# B&R Automation Studio project Huitong_FrontEval
Automation Studio 6.5.0.306; technology packages: mappView 6.5.0, OpcUaCs 6.0.0

## Configuration Config1

CPU X20CP3687X, AutomationRuntime 6.5.1, Build 11.3.0, Vc 6.0.0

### Task classes (Cpu.sw)
```
Cyclic#2:
  MidTrans <- Middleware.MidTrans.prg
Cyclic#4:
  SVG <- SVG.prg
Binaries: FWRules, mvLoader, mvConfig, udbdef, TCData, iomap, UaCsConfig, BRRole, sysconf, asfw, User, arconfig, ashwd, Role, ashwac
Libraries: AsBrStr, ArSsl, FileIO, AsARCfg, runtime, standard
```

### Hardware
```
X20CP3687X : X20CP3687X v1.9.0.0
  Connector IF2:
    ActivateDevice = 1
    Mode = Manual
    InternetAddress = 192.168.50.233
    SubnetMask = 255.255.255.0
    ActivateSnmp = 2
  ConfigurationID = Huitong_FrontEval_Config1
  Simulation = 1
  FileDevice1
  FileDeviceName1 = USER
  FileDevicePath1 = USER_PATH
  ActivateFtpServer = 1
  FTPProtocol = 1
  FtpUser1
  FtpUsername1 = br
  FtpUserPassword1 = Vr55dmG4DfTukFxBuZ2vPJZUQAb9yWCctBfVGawW8Bk=  // 123456
  FtpUserSalt1 = kenBVaZZ
  FTPAccessRight1 = 0
  ActivateWebServer = 1
  WebServerProtocol = 1
  WebServerPort = 82
  WebServerWebDir = CFCARD\WEBROOT\
  WebServerStartPage = color01.html
  WebServerAspActivate = 1
  WebServerAspReadOnly = 0
  ActivateSdm = 1
```

## Configuration x1685

CPU X20CP1685, AutomationRuntime 6.5.1, Build 11.3.0, Vc 6.0.0

### Task classes (Cpu.sw)
```
Cyclic#2:
  MidTrans <- Middleware.MidTrans.prg
Cyclic#3:
  LQR <- LQR.prg
Cyclic#4:
  SVG <- SVG.prg
Cyclic#5:
  HmiBridge <- Middleware.HmiBridge.prg
Binaries: FWRules, mvLoader, mvConfig, udbdef, TCData, iomap, UaCsConfig, BRRole, sysconf, asfw, User, arconfig, ashwd, Role, ashwac
Libraries: AsBrStr, ArSsl, FileIO, AsARCfg, runtime, standard
```

### Hardware
```
X20CP1685 : X20CP1685 v1.9.0.0
  Connector IF2:
    ActivateDevice = 1
    Mode = Manual
    InternetAddress = 192.168.50.222
    SubnetMask = 255.255.255.0
    ActivateSnmp = 2
  Connector IF3:
    CycleTime = 400
  ConfigurationID = Huitong_FrontEval_Config1
  FileDevice1
  FileDeviceName1 = USER
  FileDevicePath1 = USER_PATH
  ActivateFtpServer = 1
  FTPProtocol = 1
  FtpUser1
  FtpUsername1 = br
  FtpUserPassword1 = Vr55dmG4DfTukFxBuZ2vPJZUQAb9yWCctBfVGawW8Bk=  // 123456
  FtpUserSalt1 = kenBVaZZ
  FTPAccessRight1 = 0
  ActivateWebServer = 1
  WebServerProtocol = 1
  WebServerPort = 82
  WebServerWebDir = CFCARD\WEBROOT\
  WebServerStartPage = color01.html
  WebServerAspActivate = 1
  WebServerAspReadOnly = 0
  ActivateSdm = 1
```

## Configuration x3687x

### Task classes (Cpu.sw)
```
Cyclic#2:
  MidTrans <- Middleware.MidTrans.prg
Cyclic#3:
  LQR <- LQR.prg
Cyclic#4:
  SVG <- SVG.prg
Binaries: FWRules, mvLoader, mvConfig, udbdef, TCData, iomap, UaCsConfig, BRRole, sysconf, asfw, User, arconfig, ashwd, Role, ashwac
Libraries: AsBrStr, ArSsl, FileIO, AsARCfg, runtime, standard
```

### Hardware
```
X20CP3687X : X20CP3687X v1.9.0.0
  Connector IF2:
    ActivateDevice = 1
    Mode = Manual
    InternetAddress = 192.168.50.233
    SubnetMask = 255.255.255.0
    ActivateSnmp = 2
  ConfigurationID = Huitong_FrontEval_Config1
  FileDevice1
  FileDeviceName1 = USER
  FileDevicePath1 = USER_PATH
  ActivateFtpServer = 1
  FTPProtocol = 1
  FtpUser1
  FtpUsername1 = br
  FtpUserPassword1 = Vr55dmG4DfTukFxBuZ2vPJZUQAb9yWCctBfVGawW8Bk=  // 123456
  FtpUserSalt1 = kenBVaZZ
  FTPAccessRight1 = 0
  ActivateWebServer = 1
  WebServerProtocol = 1
  WebServerPort = 82
  WebServerWebDir = CFCARD\WEBROOT\
  WebServerStartPage = color01.html
  WebServerAspActivate = 1
  WebServerAspReadOnly = 0
  ActivateSdm = 1
```

## Logical view

Binary libraries used (declarations not repeated): operator, runtime, AsIecCon, AsBrStr, AsARCfg, standard

### Package Logical/Libraries - Global libraries

- Visualisation Logical/mappView (not shown)

### Program Logical/Middleware/MidTrans (ANSIC)

#### Main.c - Init, cyclic, exit code
```c
#include <bur/plctypes.h>

#include <stdio.h>
#include <stdint.h>
#include <string.h>
#include <math.h>

#include "Function.h"

#define SIN_DATA_LENGTH 1000
#define SIN_AMPLITUDE 127.5
#define SIN_OFFSET 127.5
#define MAX_UDINT 4294967295U

#ifdef _DEFAULT_INCLUDES
	#include <AsDefault.h>
#endif

void _INIT ProgramInit(void)
{
	gstHmi.stInputs.diLockBoxWidth = 40;
	gstMainInface.stFromMain.diSImage = 600;
	gstMainInface.stToMain.usiActivePU = 0;
	brsstrcpy((UDINT)gstHmi.stConfig.strPuChartAdr, (UDINT)&"http://");

	/********************计算IP**************************/
	fbCfgGetIPAddr.enable = 1;
	fbCfgGetIPAddr.pDevice = (UDINT)&"IF2";
	fbCfgGetIPAddr.pIPAddr = (UDINT)strTemp;
	fbCfgGetIPAddr.Len = sizeof(strTemp);
	CfgGetIPAddr(&fbCfgGetIPAddr);

	brsstrcat((UDINT)gstHmi.stConfig.strPuChartAdr, (UDINT)strTemp);
	bSimTemp = 1;
}

void _CYCLIC ProgramCyclic(void)
{
	/**********************************以下为临时程序***************************************************/
	if(1 == bSimTemp) {
		/********************** 模拟仿真数据生成 ***************************/
		if(0 == stOldHmiInput.bRefreshSimData && 1 == gstHmi.stInputs.bRefreshSimData) {
			for(udiIdx = 0; udiIdx < ST_DATA_LEN; udiIdx++) {
				rSinValue = sin(2.0 * 3.14159265358979 * (REAL)(udiSinPhase + udiIdx) / 1000.0);
				gstMainInface.stFromMain.usiDataST1[udiIdx] = (USINT)(rSinValue * SIN_AMPLITUDE + SIN_OFFSET);

				rSinValue = sin(2.0 * 3.14159265358979 * (REAL)(udiSinPhase + udiIdx + 250) / 1000.0);
				gstMainInface.stFromMain.usiDataST2[udiIdx] = (USINT)(rSinValue * SIN_AMPLITUDE + SIN_OFFSET);

				rSinValue = sin(2.0 * 3.14159265358979 * (REAL)(udiSinPhase + udiIdx + 500) / 1000.0);
				gstMainInface.stFromMain.usiDataST3[udiIdx] = (USINT)(rSinValue * SIN_AMPLITUDE + SIN_OFFSET);

				rSinValue = sin(2.0 * 3.14159265358979 * (REAL)(udiSinPhase + udiIdx + 750) / 1000.0);
				gstMainInface.stFromMain.usiDataST4[udiIdx] = (USINT)(rSinValue * SIN_AMPLITUDE + SIN_OFFSET);

				rSinValue = sin(2.0 * 3.14159265358979 * (REAL)(udiSinPhase + udiIdx + 1000) / 1000.0);
				gstMainInface.stFromMain.usiDataST5[udiIdx] = (USINT)(rSinValue * SIN_AMPLITUDE + SIN_OFFSET);

				rSinValue = sin(2.0 * 3.14159265358979 * (REAL)(udiSinPhase + udiIdx + 1250) / 1000.0);
				gstMainInface.stFromMain.usiDataST6[udiIdx] = (USINT)(rSinValue * SIN_AMPLITUDE + SIN_OFFSET);
			}
		}

		if(0 == stOldHmiInput.bMoveCurveLeft && 1 == gstHmi.stInputs.bMoveCurveLeft) {
			for(udiIdx = 0; udiIdx < ST_DATA_LEN; udiIdx++) {
				rSinValue = sin(2.0 * 3.14159265358979 * (REAL)(udiSinPhase + udiIdx) / 1000.0);
				gstMainInface.stFromMain.usiDataST1[udiIdx] = (USINT)(rSinValue * SIN_AMPLITUDE + SIN_OFFSET);

				rSinValue = sin(2.0 * 3.14159265358979 * (REAL)(udiSinPhase + udiIdx + 250) / 1000.0);
				gstMainInface.stFromMain.usiDataST2[udiIdx] = (USINT)(rSinValue * SIN_AMPLITUDE + SIN_OFFSET);

				rSinValue = sin(2.0 * 3.14159265358979 * (REAL)(udiSinPhase + udiIdx + 500) / 1000.0);
				gstMainInface.stFromMain.usiDataST3[udiIdx] = (USINT)(rSinValue * SIN_AMPLITUDE + SIN_OFFSET);

				rSinValue = sin(2.0 * 3.14159265358979 * (REAL)(udiSinPhase + udiIdx + 750) / 1000.0);
				gstMainInface.stFromMain.usiDataST4[udiIdx] = (USINT)(rSinValue * SIN_AMPLITUDE + SIN_OFFSET);

				rSinValue = sin(2.0 * 3.14159265358979 * (REAL)(udiSinPhase + udiIdx + 1000) / 1000.0);
				gstMainInface.stFromMain.usiDataST5[udiIdx] = (USINT)(rSinValue * SIN_AMPLITUDE + SIN_OFFSET);

				rSinValue = sin(2.0 * 3.14159265358979 * (REAL)(udiSinPhase + udiIdx + 1250) / 1000.0);
				gstMainInface.stFromMain.usiDataST6[udiIdx] = (USINT)(rSinValue * SIN_AMPLITUDE + SIN_OFFSET);
			}

			udiSinPhase -= 100;
			if(udiSinPhase <= 0) {
				udiSinPhase = 1000;
			}
		}

		if(0 == stOldHmiInput.bMoveCurveRight && 1 == gstHmi.stInputs.bMoveCurveRight) {
			for(udiIdx = 0; udiIdx < ST_DATA_LEN; udiIdx++) {
				rSinValue = sin(2.0 * 3.14159265358979 * (REAL)(udiSinPhase + udiIdx) / 1000.0);
				gstMainInface.stFromMain.usiDataST1[udiIdx] = (USINT)(rSinValue * SIN_AMPLITUDE + SIN_OFFSET);

				rSinValue = sin(2.0 * 3.14159265358979 * (REAL)(udiSinPhase + udiIdx + 250) / 1000.0);
				gstMainInface.stFromMain.usiDataST2[udiIdx] = (USINT)(rSinValue * SIN_AMPLITUDE + SIN_OFFSET);

				rSinValue = sin(2.0 * 3.14159265358979 * (REAL)(udiSinPhase + udiIdx + 500) / 1000.0);
				gstMainInface.stFromMain.usiDataST3[udiIdx] = (USINT)(rSinValue * SIN_AMPLITUDE + SIN_OFFSET);

				rSinValue = sin(2.0 * 3.14159265358979 * (REAL)(udiSinPhase + udiIdx + 750) / 1000.0);
				gstMainInface.stFromMain.usiDataST4[udiIdx] = (USINT)(rSinValue * SIN_AMPLITUDE + SIN_OFFSET);

				rSinValue = sin(2.0 * 3.14159265358979 * (REAL)(udiSinPhase + udiIdx + 1000) / 1000.0);
				gstMainInface.stFromMain.usiDataST5[udiIdx] = (USINT)(rSinValue * SIN_AMPLITUDE + SIN_OFFSET);

				rSinValue = sin(2.0 * 3.14159265358979 * (REAL)(udiSinPhase + udiIdx + 1250) / 1000.0);
				gstMainInface.stFromMain.usiDataST6[udiIdx] = (USINT)(rSinValue * SIN_AMPLITUDE + SIN_OFFSET);
			}

			udiSinPhase += 100;
			if(udiSinPhase >= 1000) {
				udiSinPhase = 0;
			}
		}

		// (Temp) 当前横向自定义距离值，计算
		if(0 == stOldHmiInput.bVisMarkIntervalMinus && 1 == gstHmi.stInputs.bVisMarkIntervalMinus) {
			gstMainInface.stFromMain.diPuWindowIntervalmm = gstMainInface.stFromMain.diPuWindowIntervalmm - 20;
		}

		if(0 == stOldHmiInput.bVisMarkIntervalAdd && 1 == gstHmi.stInputs.bVisMarkIntervalAdd) {
			gstMainInface.stFromMain.diPuWindowIntervalmm = gstMainInface.stFromMain.diPuWindowIntervalmm + 20;
		}
		// 锁标窗口左移与右移动控制，锁定功能
		// 锁定
		if (0 == stOldHmiInput.bCmdLatchPos && 1 == gstHmi.stInputs.bCmdLatchPos) {
			if (gstMainInface.stFromMain.usiActiveDrawMode == 10 || gstMainInface.stFromMain.usiActiveDrawMode == 11) {
				gstMainInface.stFromMain.udiActivePuLatchPos = cal_LatchPos(gstHmi.stInputs.iSelectFront, gstHmi.stInputs.iSelectFirst, gstMainInface.stFromMain.diSImage*1000, gstAspInface.stFromAsp.udiCurLatchPosition);
			} else {
				gstMainInface.stFromMain.udiActivePuLatchPos = gstAspInface.stFromAsp.udiCurLatchPosition;
			}
		}
		// 右移
		if (0 == stOldHmiInput.bMoveLockBoxRight && 1 == gstHmi.stInputs.bMoveLockBoxRight) {
			gstMainInface.stFromMain.udiActivePuLatchPos = gstMainInface.stFromMain.udiActivePuLatchPos + 1000;
		}
		// 左移
		if (0 == stOldHmiInput.bMoveLockBoxLeft && 1 == gstHmi.stInputs.bMoveLockBoxLeft) {
			gstMainInface.stFromMain.udiActivePuLatchPos = gstMainInface.stFromMain.udiActivePuLatchPos - 1000;

		}
		// 限幅
		if (gstMainInface.stFromMain.udiActivePuLatchPos > (UDINT)gstMainInface.stFromMain.diSImage * 1000) {
			gstMainInface.stFromMain.udiActivePuLatchPos = (UDINT)gstMainInface.stFromMain.diSImage * 1000;
		}
		if (gstMainInface.stFromMain.udiActivePuLatchPos < 0) {
			gstMainInface.stFromMain.udiActivePuLatchPos = 0;
		}

		// 计算BST锁标偏移
		if (gstMainInface.stFromMain.usiActiveDrawMode == 10 || gstMainInface.stFromMain.usiActiveDrawMode == 11) {
			cal_BST_Idx(gstHmi.stInputs.iSelectFront, gstHmi.stInputs.iSelectFirst, 0, &gstMainInface.stFromMain.usiMarkSelectFront, &gstMainInface.stFromMain.usiMarkSelectFirst, &gstMainInface.stFromMain.usiMarkSelectSelf);

		}
	}
	/*******************************临时程序到此为止*****************************************************/

	/********************** 色组选择换算 ***************************/
	// gstMiddle.stOutputs.diPuNum
	for(udiIdx = 0; udiIdx < sizeof(gstHmi.stInputs.bCheckedPu)/sizeof(gstHmi.stInputs.bCheckedPu[0]); udiIdx ++) {
		if (1 == gstHmi.stInputs.bCheckedPu[udiIdx] && 0 == stOldHmiInput.bCheckedPu[udiIdx]) {
			brsmemset((UDINT)gstHmi.stInputs.bCheckedPu,0 , sizeof(gstHmi.stInputs.bCheckedPu));
			gstMainInface.stToMain.usiActivePU = (USINT)udiIdx;
		}
	}
	/********************** 绘图数据转换 ***************************/

	if (0 == gstMainInface.stFromMain.usiActiveDrawMode || 1 == gstMainInface.stFromMain.usiActiveDrawMode) {
		// 1号传感器数据
		uint8_to_base64_string(gstMainInface.stFromMain.usiDataST1, ST_DATA_LEN, strHexStrBuffer);
		// bytes_to_hex_string(gstMainInface.stFromMain.usiDataST1, ST_DATA_LEN, strHexStrBuffer);
		for(udiIdx = 0; udiIdx < ST_SEP_LEN; udiIdx ++) {
			brsmemcpy((UDINT)gstAspInface.stToAsp.strDataST1[udiIdx] , (UDINT)&strHexStrBuffer[ST_SEP_DATA_LEN * udiIdx], ST_SEP_DATA_LEN);
		}
		// 2号传感器数据
		uint8_to_base64_string(gstMainInface.stFromMain.usiDataST2, ST_DATA_LEN, strHexStrBuffer);
		// bytes_to_hex_string(gstMainInface.stFromMain.usiDataST2, ST_DATA_LEN, strHexStrBuffer);
		for(udiIdx = 0; udiIdx < ST_SEP_LEN; udiIdx ++) {
			brsmemcpy((UDINT)gstAspInface.stToAsp.strDataST2[udiIdx] , (UDINT)&strHexStrBuffer[ST_SEP_DATA_LEN * udiIdx], ST_SEP_DATA_LEN);
		}
		// 3 号传感器数据
		for(udiIdx = 0; udiIdx < ST_SEP_LEN; udiIdx ++) {
			gstAspInface.stToAsp.strDataST3[udiIdx][0] = '\0';
		}
		// 4 号传感器数据
		for(udiIdx = 0; udiIdx < ST_SEP_LEN; udiIdx ++) {
			gstAspInface.stToAsp.strDataST4[udiIdx][0] = '\0';
		}
		// 5 号传感器数据
		for(udiIdx = 0; udiIdx < ST_SEP_LEN; udiIdx ++) {
			gstAspInface.stToAsp.strDataST5[udiIdx][0] = '\0';
		}
		// 6 号传感器数据
		for(udiIdx = 0; udiIdx < ST_SEP_LEN; udiIdx ++) {
			gstAspInface.stToAsp.strDataST6[udiIdx][0] = '\0';
		}
	} 	else if(2 == gstMainInface.stFromMain.usiActiveDrawMode) {
		// 1号传感器数据
		uint8_to_base64_string(gstMainInface.stFromMain.usiDataST1, ST_DATA_LEN, strHexStrBuffer);
		for(udiIdx = 0; udiIdx < ST_SEP_LEN; udiIdx ++) {
			brsmemcpy((UDINT)gstAspInface.stToAsp.strDataST1[udiIdx] , (UDINT)&strHexStrBuffer[ST_SEP_DATA_LEN * udiIdx], ST_SEP_DATA_LEN);
		}
		// 2 号传感器数据
		for(udiIdx = 0; udiIdx < ST_SEP_LEN; udiIdx ++) {
			gstAspInface.stToAsp.strDataST2[udiIdx][0] = '\0';
		}
		// 3 号传感器数据
		for(udiIdx = 0; udiIdx < ST_SEP_LEN; udiIdx ++) {
			gstAspInface.stToAsp.strDataST3[udiIdx][0] = '\0';
		}
		// 4 号传感器数据
		for(udiIdx = 0; udiIdx < ST_SEP_LEN; udiIdx ++) {
			gstAspInface.stToAsp.strDataST4[udiIdx][0] = '\0';
		}
		// 5 号传感器数据
		for(udiIdx = 0; udiIdx < ST_SEP_LEN; udiIdx ++) {
			gstAspInface.stToAsp.strDataST5[udiIdx][0] = '\0';
		}
		// 6 号传感器数据
		for(udiIdx = 0; udiIdx < ST_SEP_LEN; udiIdx ++) {
			gstAspInface.stToAsp.strDataST6[udiIdx][0] = '\0';
		}
	} 	else if (3 == gstMainInface.stFromMain.usiActiveDrawMode) {
		// 1 号传感器数据
		for(udiIdx = 0; udiIdx < ST_SEP_LEN; udiIdx ++) {
			gstAspInface.stToAsp.strDataST1[udiIdx][0] = '\0';
		}
		// 2 号传感器数据
		uint8_to_base64_string(gstMainInface.stFromMain.usiDataST2, ST_DATA_LEN, strHexStrBuffer);
		for(udiIdx = 0; udiIdx < ST_SEP_LEN; udiIdx ++) {
			brsmemcpy((UDINT)gstAspInface.stToAsp.strDataST2[udiIdx] , (UDINT)&strHexStrBuffer[ST_SEP_DATA_LEN * udiIdx], ST_SEP_DATA_LEN);
		}
		// 3 号传感器数据
		for(udiIdx = 0; udiIdx < ST_SEP_LEN; udiIdx ++) {
			gstAspInface.stToAsp.strDataST3[udiIdx][0] = '\0';
		}
		// 4 号传感器数据
		for(udiIdx = 0; udiIdx < ST_SEP_LEN; udiIdx ++) {
			gstAspInface.stToAsp.strDataST4[udiIdx][0] = '\0';
		}
		// 5 号传感器数据
		for(udiIdx = 0; udiIdx < ST_SEP_LEN; udiIdx ++) {
			gstAspInface.stToAsp.strDataST5[udiIdx][0] = '\0';
		}
		// 6号传感器数据
		for(udiIdx = 0; udiIdx < ST_SEP_LEN; udiIdx ++) {
			gstAspInface.stToAsp.strDataST6[udiIdx][0] = '\0';
		}
	} else if (10 == gstMainInface.stFromMain.usiActiveDrawMode || 11 == gstMainInface.stFromMain.usiActiveDrawMode) {
		// 1号传感器数据
		uint8_to_base64_string(gstMainInface.stFromMain.usiDataST1, ST_DATA_LEN, strHexStrBuffer);
		for(udiIdx = 0; udiIdx < ST_SEP_LEN; udiIdx ++) {
			brsmemcpy((UDINT)gstAspInface.stToAsp.strDataST1[udiIdx] , (UDINT)&strHexStrBuffer[ST_SEP_DATA_LEN * udiIdx], ST_SEP_DATA_LEN);
		}
		// 2号传感器数据
		uint8_to_base64_string(gstMainInface.stFromMain.usiDataST2, ST_DATA_LEN, strHexStrBuffer);
		for(udiIdx = 0; udiIdx < ST_SEP_LEN; udiIdx ++) {
			brsmemcpy((UDINT)gstAspInface.stToAsp.strDataST2[udiIdx] , (UDINT)&strHexStrBuffer[ST_SEP_DATA_LEN * udiIdx], ST_SEP_DATA_LEN);
		}
		// 3号传感器数据
		uint8_to_base64_string(gstMainInface.stFromMain.usiDataST3, ST_DATA_LEN, strHexStrBuffer);
		for(udiIdx = 0; udiIdx < ST_SEP_LEN; udiIdx ++) {
			brsmemcpy((UDINT)gstAspInface.stToAsp.strDataST3[udiIdx] , (UDINT)&strHexStrBuffer[ST_SEP_DATA_LEN * udiIdx], ST_SEP_DATA_LEN);
		}
		// 4号传感器数据
		uint8_to_base64_string(gstMainInface.stFromMain.usiDataST4, ST_DATA_LEN, strHexStrBuffer);
		for(udiIdx = 0; udiIdx < ST_SEP_LEN; udiIdx ++) {
			brsmemcpy((UDINT)gstAspInface.stToAsp.strDataST4[udiIdx] , (UDINT)&strHexStrBuffer[ST_SEP_DATA_LEN * udiIdx], ST_SEP_DATA_LEN);
		}
		// 5号传感器数据
		uint8_to_base64_string(gstMainInface.stFromMain.usiDataST5, ST_DATA_LEN, strHexStrBuffer);
		for(udiIdx = 0; udiIdx < ST_SEP_LEN; udiIdx ++) {
			brsmemcpy((UDINT)gstAspInface.stToAsp.strDataST5[udiIdx] , (UDINT)&strHexStrBuffer[ST_SEP_DATA_LEN * udiIdx], ST_SEP_DATA_LEN);
		}
		// 6号传感器数据
		uint8_to_base64_string(gstMainInface.stFromMain.usiDataST6, ST_DATA_LEN, strHexStrBuffer);
		for(udiIdx = 0; udiIdx < ST_SEP_LEN; udiIdx ++) {
			brsmemcpy((UDINT)gstAspInface.stToAsp.strDataST6[udiIdx] , (UDINT)&strHexStrBuffer[ST_SEP_DATA_LEN * udiIdx], ST_SEP_DATA_LEN);
		}
	} else {
		// 1 号传感器数据
		for(udiIdx = 0; udiIdx < ST_SEP_LEN; udiIdx ++) {
			gstAspInface.stToAsp.strDataST1[udiIdx][0] = '\0';
		}
		// 2 号传感器数据
		for(udiIdx = 0; udiIdx < ST_SEP_LEN; udiIdx ++) {
			gstAspInface.stToAsp.strDataST2[udiIdx][0] = '\0';
		}
		// 3 号传感器数据
		for(udiIdx = 0; udiIdx < ST_SEP_LEN; udiIdx ++) {
			gstAspInface.stToAsp.strDataST3[udiIdx][0] = '\0';
		}
		// 4 号传感器数据
		for(udiIdx = 0; udiIdx < ST_SEP_LEN; udiIdx ++) {
			gstAspInface.stToAsp.strDataST4[udiIdx][0] = '\0';
		}
		// 5 号传感器数据
		for(udiIdx = 0; udiIdx < ST_SEP_LEN; udiIdx ++) {
			gstAspInface.stToAsp.strDataST5[udiIdx][0] = '\0';
		}
		// 6 号传感器数据
		for(udiIdx = 0; udiIdx < ST_SEP_LEN; udiIdx ++) {
			gstAspInface.stToAsp.strDataST6[udiIdx][0] = '\0';
		}
	}

	/********************** 编码器数据生成 ***************************/
	for (udiIdx = 0; udiIdx < ST_PU_SIZE; udiIdx++) {
		gstHmi.stOutputs.rPuBiasValue[udiIdx] = random_real(-5.0, 5.0);
		gstHmi.stOutputs.rPuBiasHigh[udiIdx] = 20.0;
		gstHmi.stOutputs.rPuBiasLow[udiIdx] = -20.0;
	}

	/********************** 与ASP层的通信交互 ***************************/
	gstAspInface.stToAsp.udiCurLatchPosition   = gstMainInface.stFromMain.udiActivePuLatchPos;
	gstAspInface.stToAsp.usiCmdLatchPos        = (USINT)gstHmi.stInputs.bCmdLatchPos;
	gstAspInface.stToAsp.diWindowWidth         = gstHmi.stInputs.diLockBoxWidth;
	gstAspInface.stToAsp.diPuWindowIntervalmm  = gstMainInface.stFromMain.diPuWindowIntervalmm;
	gstAspInface.stToAsp.usiActiveDrawMode	   = gstMainInface.stFromMain.usiActiveDrawMode;
	gstAspInface.stToAsp.diSImage			   = gstMainInface.stFromMain.diSImage;

	// BST 标记位置计算
	if ((0 == stOldHmiInput.bCmdLatchPos && 1 == gstHmi.stInputs.bCmdLatchPos)
		&& (gstMainInface.stFromMain.usiActiveDrawMode == 10 || gstMainInface.stFromMain.usiActiveDrawMode == 11)) {
		if (gstHmi.stInputs.bMarkSelectSelfEnable) {
			gstAspInface.stToAsp.udiMarkSelfPosition =
			(gstMainInface.stFromMain.udiActivePuLatchPos + (UDINT)gstMainInface.stFromMain.usiMarkSelectSelf  * BST_SEG_UM) % (UDINT)(gstMainInface.stFromMain.diSImage * 1000);
		}else {
			gstAspInface.stToAsp.udiMarkSelfPosition = MAX_UDINT;
		}

		if (gstHmi.stInputs.bMarkSelectFirstEnable) {
			gstAspInface.stToAsp.udiMarkFirstPosition =
			(gstMainInface.stFromMain.udiActivePuLatchPos + (UDINT)gstMainInface.stFromMain.usiMarkSelectFirst * BST_SEG_UM) % (UDINT)(gstMainInface.stFromMain.diSImage * 1000);
		}else {
			gstAspInface.stToAsp.udiMarkFirstPosition = MAX_UDINT;
		}

		if (gstHmi.stInputs.bMarkSelectFrontEnable) {
			gstAspInface.stToAsp.udiMarkFrontPosition =
			(gstMainInface.stFromMain.udiActivePuLatchPos + (UDINT)gstMainInface.stFromMain.usiMarkSelectFront * BST_SEG_UM) % (UDINT)(gstMainInface.stFromMain.diSImage * 1000);
		}else {
			gstAspInface.stToAsp.udiMarkFrontPosition = MAX_UDINT;
		}
	}

	// 计算 usiMarkEnableBST：按位操作
	// 最低位 (Bit 0) 对应 Self (bMarkSelectSelfEnable)
	// 次低位 (Bit 1) 对应 Front (bMarkSelectFrontEnable)
	// 第 2 位 (Bit 2) 对应 First (bMarkSelectFirstEnable)
	gstAspInface.stToAsp.usiMarkEnableBST = 0;
	if (gstHmi.stInputs.bMarkSelectSelfEnable) {
		gstAspInface.stToAsp.usiMarkEnableBST |= 0x01; // Set Bit 0
	}
	if (gstHmi.stInputs.bMarkSelectFrontEnable) {
		gstAspInface.stToAsp.usiMarkEnableBST |= 0x02; // Set Bit 1
	}
	if (gstHmi.stInputs.bMarkSelectFirstEnable) {
		gstAspInface.stToAsp.usiMarkEnableBST |= 0x04; // Set Bit 2
	}

	/********************** 与主控的通信交互 ***************************/
	gstMainInface.stToMain.usiCmdLatchPos      = (USINT)gstHmi.stInputs.bCmdLatchPos;
	gstMainInface.stToMain.diWindowWidth       = gstHmi.stInputs.diLockBoxWidth;
	gstMainInface.stToMain.usiCmdLeft          = (USINT)gstHmi.stInputs.bMoveCurveLeft;
	gstMainInface.stToMain.usiCmdRight         = (USINT)gstHmi.stInputs.bMoveCurveRight;
	gstMainInface.stToMain.usiCmdLatchPosLeft  = (USINT)gstHmi.stInputs.bMoveLockBoxLeft;
	gstMainInface.stToMain.usiCmdLatchPosRight = (USINT)gstHmi.stInputs.bMoveLockBoxRight;
	gstMainInface.stToMain.usiVisMarkIntervalAdd   = (USINT)gstHmi.stInputs.bVisMarkIntervalAdd;
	gstMainInface.stToMain.usiVisMarkIntervalMinus = (USINT)gstHmi.stInputs.bVisMarkIntervalMinus;
	gstMainInface.stToMain.usiActivePuTeachMode = (USINT)gstHmi.stInputs.bActivePuTeachMode;
	gstMainInface.stFromMain.usiActiveDrawMode;  // 绘图模式

	// 触发锁标按钮后，将Asp读取到的位置
	if (0 == stOldHmiInput.bCmdLatchPos && 1 == gstHmi.stInputs.bCmdLatchPos) {
		gstMainInface.stToMain.udiLatchPosition[gstMainInface.stToMain.usiActivePU] = gstAspInface.stFromAsp.udiCurLatchPosition;
		if (gstMainInface.stFromMain.usiActiveDrawMode == 10 || gstMainInface.stFromMain.usiActiveDrawMode == 11) {

			gstMainInface.stToMain.udiLatchPosition[gstMainInface.stToMain.usiActivePU] = gstAspInface.stFromAsp.udiCurLatchPosition
				+ (UDINT)(find_min_of_three(gstHmi.stInputs.iSelectFront, gstHmi.stInputs.iSelectFirst, 0) * (INT)BST_SEG_UM);
		}
	}

	gstHmi.stOutputs.diSImage = gstMainInface.stFromMain.diSImage;
	gstHmi.stOutputs.diPuWindowIntervalmm = gstMainInface.stFromMain.diPuWindowIntervalmm;

	/********************** Old ***************************/
	brsmemcpy((UDINT)&stOldHmiInput, (UDINT)&gstHmi.stInputs, sizeof(gstHmi.stInputs));

}

void _EXIT ProgramExit(void)
{

}
```

#### Function.c - Function
```c
#include "Function.h"
#include <stdlib.h>
#include <string.h>

/* HEX 编码 */
void byte_to_hex_str(uint8_t byte, char* out) {
	const char hex_chars[] = "0123456789ABCDEF";
	out[0] = hex_chars[(byte >> 4) & 0x0F];
	out[1] = hex_chars[byte & 0x0F];
}

void bytes_to_hex_string(const uint8_t* input, size_t len, char* output) {
	for (size_t i = 0; i < len; ++i) {
		byte_to_hex_str(input[i], output + i * 2);
	}
	output[len * 2] = '\0';
}

/* BASE64 编码 */
static const char base64_table[] = "ABCDEFGHIJKLMNOPQRSTUVWXYZabcdefghijklmnopqrstuvwxyz0123456789+/";

int uint8_to_base64_string(const uint8_t *input, int input_len, char *output) {
	int i = 0;
	int out_idx = 0;

	while (i < input_len - 2) {
		uint8_t b0 = input[i];
		uint8_t b1 = input[i+1];
		uint8_t b2 = input[i+2];

		output[out_idx++] = base64_table[b0 >> 2];
		output[out_idx++] = base64_table[((b0 & 0x03) << 4) | (b1 >> 4)];
		output[out_idx++] = base64_table[((b1 & 0x0F) << 2) | (b2 >> 6)];
		output[out_idx++] = base64_table[b2 & 0x3F];

		i += 3;
	}

	if (i < input_len) {
		uint8_t b0 = input[i];
		uint8_t b1 = input[i+1];

		output[out_idx++] = base64_table[b0 >> 2];
		output[out_idx++] = base64_table[((b0 & 0x03) << 4) | (b1 >> 4)];
		output[out_idx++] = '=';
		output[out_idx++] = '=';
	} else if (i == input_len - 1) {
		uint8_t b0 = input[i];

		output[out_idx++] = base64_table[b0 >> 2];
		output[out_idx++] = base64_table[(b0 & 0x03) << 4];
		output[out_idx++] = '=';
		output[out_idx++] = '=';
	}

	output[out_idx] = '\0';

	return out_idx;
}

INT find_min_of_three(INT val1, INT val2, INT val3) {
	INT min_val = val1;

	if (val2 < min_val) {
		min_val = val2;
	}
	if (val3 < min_val) {
		min_val = val3;
	}

	return min_val;
}

INT cal_BST_Idx(INT val1, INT val2, INT val3, USINT* out1, USINT* out2, USINT* out3) {
	INT min_val = val1;
	min_val = find_min_of_three(val1, val2, val3);
	INT offset = 0;
	if (min_val < 0) {
		offset = -min_val;
	}

	*out1 = (USINT)(val1 + offset);
	*out2 = (USINT)(val2 + offset);
	*out3 = (USINT)(val3 + offset);

	return offset;
}

UDINT cal_LatchPos(INT idx1, INT idx2, DINT diSImage, UDINT CurLatchPos) {
	INT minIdx = find_min_of_three(idx1, idx2, 0);

	DINT offset = (DINT)minIdx * (DINT)BST_SEG_UM;

	DINT tempPos = (DINT)CurLatchPos + offset;

	DINT maxLimit = (DINT)diSImage;

	if (tempPos < 0) {
		DINT cycles = (-tempPos) / (maxLimit + 1) + 1;
		tempPos += cycles * (maxLimit + 1);
	}

	tempPos = tempPos % (maxLimit + 1);

	if (tempPos < 0) {
		tempPos = 0;
	}
	return (UDINT)tempPos;
}

REAL random_real(REAL rMin, REAL rMax) {
	REAL lo = rMin;
	REAL hi = rMax;
	REAL t;

	if (hi < lo) {
		REAL tmp = lo;
		lo = hi;
		hi = tmp;
	}

	if (lo == hi) {
		return lo;
	}

	t = (REAL)rand() / ((REAL)RAND_MAX + 1.0f);
	return lo + t * (hi - lo);
}
```

#### Function.h - Function
```c
#ifndef MIDTRANS_FUNCTION_H
#define MIDTRANS_FUNCTION_H

#include <bur/plctypes.h>
#include <stddef.h>

#define uint8_t USINT
#define BST_SEG_UM 20000U

void byte_to_hex_str(uint8_t byte, char* out);
void bytes_to_hex_string(const uint8_t* input, size_t len, char* output);
int uint8_to_base64_string(const uint8_t *input, int input_len, char *output);
INT find_min_of_three(INT val1, INT val2, INT val3);
INT cal_BST_Idx(INT val1, INT val2, INT val3, USINT* out1, USINT* out2, USINT* out3);
UDINT cal_LatchPos(INT idx1, INT idx2, DINT diSImage, UDINT CurLatchPos);
REAL random_real(REAL rMin, REAL rMax);

#endif
```

#### Variables.var - Local variables
```iecst
VAR
	udiIdx : UDINT;
	strHexStrBuffer : STRING[ST_DATA_LEN_DOUBLE];
	stOldHmiInput : HMI_Input_typ;
	rSinValue : REAL;
	udiSinPhase : UDINT;
	bSimTemp : BOOL;
	fbCfgGetIPAddr : CfgGetIPAddr;
	strTemp : STRING[32];
END_VAR
```

### Program Logical/Middleware/HmiBridge (ANSIC)

#### Main.c - Init, cyclic, exit code
```c
#include <bur/plctypes.h>

#ifdef _DEFAULT_INCLUDES
	#include <AsDefault.h>
#endif

#include "HmiBridgeSync.h"
#include "HmiBridgeControl.h"

void _INIT ProgramInit(void)
{
	HmiBridgeInitDemoValues();
}

void _CYCLIC ProgramCyclic(void)
{
	HmiBridgeSyncRegisteredVariables();
	HmiBridgeDemoControlStep();
	HmiBridgeSyncRegisteredVariables();
}

void _EXIT ProgramExit(void)
{
}
```

#### HmiBridgeControl.h - HMI bridge control helpers
```c
#ifndef HMIBRIDGE_CONTROL_H
#define HMIBRIDGE_CONTROL_H

static REAL HmiBridgeClampReal(REAL value, REAL minValue, REAL maxValue)
{
	if (value < minValue) {
		return minValue;
	}
	if (value > maxValue) {
		return maxValue;
	}
	return value;
}

static void HmiBridgeInitDemoValues(void)
{
	HMI_MW_U00_Bridge_Cmd_EnableReq = 0;
	HMI_MW_U00_Bridge_Par_Target = 100.0f;
	HMI_MW_U00_Bridge_Par_Mode = 1;

	HMI_MW_U00_Bridge_InOut_Trim = 0.0f;
	HMI_MW_U00_Bridge_InOut_Offset = 0;
	HMI_MW_U00_Bridge_InOut_Recipe = 1;

	stHmiBridgeOld.stInOut.rTrimValue = HMI_MW_U00_Bridge_InOut_Trim;
	stHmiBridgeOld.stInOut.diSharedOffset = HMI_MW_U00_Bridge_InOut_Offset;
	stHmiBridgeOld.stInOut.usiRecipeNo = HMI_MW_U00_Bridge_InOut_Recipe;
	stHmiBridgeCtrl.stInOut = stHmiBridgeOld.stInOut;
}

static void HmiBridgeDemoControlStep(void)
{
	stHmiBridgeCtrl.stOutput.bReady = 1;
	stHmiBridgeCtrl.stOutput.bEnabledEcho = stHmiBridgeCtrl.stInput.bEnableReq;
	stHmiBridgeCtrl.stOutput.rAcceptedTarget =
		HmiBridgeClampReal(stHmiBridgeCtrl.stInput.rTargetValue, -1000.0f, 1000.0f);
	stHmiBridgeCtrl.stOutput.usiAcceptedMode = stHmiBridgeCtrl.stInput.usiModeSelect;

	if (stHmiBridgeCtrl.stOutput.bEnabledEcho) {
		stHmiBridgeCtrl.stOutput.rActualValue =
			stHmiBridgeCtrl.stOutput.rAcceptedTarget + stHmiBridgeCtrl.stInOut.rTrimValue;
	}
	else {
		stHmiBridgeCtrl.stOutput.rActualValue = 0.0f;
	}

	stHmiBridgeCtrl.stOutput.udiCycleCounter++;
}

#endif
```

#### HmiBridgeSync.h - HMI bridge sync helpers
```c
#ifndef HMIBRIDGE_SYNC_H
#define HMIBRIDGE_SYNC_H

#define HMI_TO_CTRL(clientVar, servVar) \
do {                                    \
	(servVar) = (clientVar);            \
} while (0)

#define CTRL_TO_HMI(clientVar, servVar) \
do {                                    \
	(clientVar) = (servVar);            \
} while (0)

#define READ_WRITE(clientVar, clientOld, servVar) \
do {                                              \
	if ((clientVar) != (clientOld)) {             \
		(servVar) = (clientVar);                  \
		(clientOld) = (clientVar);                \
	}                                             \
	else if ((clientVar) != (servVar)) {          \
		(clientVar) = (servVar);                  \
		(clientOld) = (servVar);                  \
	}                                             \
} while (0)

static void HmiBridgeSyncRegisteredVariables(void)
{
#define HMI_INPUT(hmiVar, ctrlVar) HMI_TO_CTRL(hmiVar, ctrlVar);
#define HMI_OUTPUT(hmiVar, ctrlVar) CTRL_TO_HMI(hmiVar, ctrlVar);
#define HMI_INOUT(hmiVar, oldVar, ctrlVar) READ_WRITE(hmiVar, oldVar, ctrlVar);

#include "HmiBridgeRegistry.def"

#undef HMI_INPUT
#undef HMI_OUTPUT
#undef HMI_INOUT
}

#endif
```

- HmiBridgeRegistry.def - HMI bridge variable registry (not shown)

#### Types.typ - Local data types
```iecst
TYPE
	HmiBridgeInput_typ : 	STRUCT
		bEnableReq : BOOL;
		rTargetValue : REAL;
		usiModeSelect : USINT;
	END_STRUCT;

	HmiBridgeOutput_typ : 	STRUCT
		bReady : BOOL;
		bEnabledEcho : BOOL;
		rAcceptedTarget : REAL;
		rActualValue : REAL;
		usiAcceptedMode : USINT;
		udiCycleCounter : UDINT;
	END_STRUCT;

	HmiBridgeInOut_typ : 	STRUCT
		rTrimValue : REAL;
		diSharedOffset : DINT;
		usiRecipeNo : USINT;
	END_STRUCT;

	HmiBridgeCtrl_typ : 	STRUCT
		stInput : HmiBridgeInput_typ;
		stOutput : HmiBridgeOutput_typ;
		stInOut : HmiBridgeInOut_typ;
	END_STRUCT;

	HmiBridgeOld_typ : 	STRUCT
		stInOut : HmiBridgeInOut_typ;
	END_STRUCT;
END_TYPE
```

#### Variables.var - Local variables
```iecst
VAR
	HMI_MW_U00_Bridge_Cmd_EnableReq : BOOL;
	HMI_MW_U00_Bridge_Par_Target : REAL;
	HMI_MW_U00_Bridge_Par_Mode : USINT;
	HMI_MW_U00_Bridge_Sts_Ready : BOOL;
	HMI_MW_U00_Bridge_Sts_Enabled : BOOL;
	HMI_MW_U00_Bridge_Act_Target : REAL;
	HMI_MW_U00_Bridge_Act_Value : REAL;
	HMI_MW_U00_Bridge_Sts_Mode : USINT;
	HMI_MW_U00_Bridge_Diag_Cycle : UDINT;
	HMI_MW_U00_Bridge_InOut_Trim : REAL;
	HMI_MW_U00_Bridge_InOut_Offset : DINT;
	HMI_MW_U00_Bridge_InOut_Recipe : USINT;
	stHmiBridgeCtrl : HmiBridgeCtrl_typ;
	stHmiBridgeOld : HmiBridgeOld_typ;
END_VAR
```

### GlobalMiddle.typ
```iecst
TYPE
	MiddleInput_typ : 	STRUCT
		diEchartLockPosition : DINT; (*ECharts 锁标位置返还	*)
	END_STRUCT;
	MiddleOutput_typ : 	STRUCT
		usiDrawingArr : ARRAY[0..ST_DATA_LEN_MINUS_ONE]OF USINT; (*绘图数组数据源*)
		diActualLockPos : DINT; (*实际锁标位置*)
		diActuralLockBoxWidth : DINT; (*实际锁标框宽度	*)
		diLockBoxOffset : DINT; (*锁标窗口偏移*)
		diPuNum : DINT;
	END_STRUCT;
	Middle_Interface_typ : 	STRUCT
		stInputs : MiddleInput_typ;
		stOutputs : MiddleOutput_typ;
	END_STRUCT;
	HMI_Input_typ : 	STRUCT
		bCheckedPu : ARRAY[0..16]OF BOOL;
		bMoveCurveLeft : BOOL; (*左平移曲线*)
		bMoveCurveRight : BOOL; (*右平移曲线*)
		bMoveLockBoxLeft : BOOL;
		bMoveLockBoxRight : BOOL;
		diLockBoxWidth : DINT;
		bCmdLatchPos : BOOL;
		bVisMarkIntervalAdd : BOOL;
		bVisMarkIntervalMinus : BOOL;
		bActivePuTeachMode : BOOL;
		bRefreshSimData : BOOL; (*刷新模拟数据（临时）*)
		iSelectFront : INT;
		iSelectFirst : INT;
		bMarkSelectSelfEnable : BOOL; (*本色有效标志*)
		bMarkSelectFrontEnable : BOOL; (*前色有效标志*)
		bMarkSelectFirstEnable : BOOL; (*首色有效标志*)
	END_STRUCT;
	HMI_Output_typ : 	STRUCT
		diSImage : DINT;
		diPuWindowIntervalmm : DINT; (*当前横向自定义距离值*)
		rPuBiasValue : ARRAY[0..ST_PU_SIZE]OF REAL;
		rPuBiasLow : ARRAY[0..ST_PU_SIZE]OF REAL;
		rPuBiasHigh : ARRAY[0..ST_PU_SIZE]OF REAL;
	END_STRUCT;
	HMI_Interface_typ : 	STRUCT
		stInputs : HMI_Input_typ; (*HMI 写入 → PLC 读取*)
		stOutputs : HMI_Output_typ; (*PLC 写入 → HMI 读取*)
		stConfig : HMI_Config_typ;
	END_STRUCT;
	HMI_Config_typ : 	STRUCT
		strPuChartAdr : STRING[80];
	END_STRUCT;
	FromAsp_typ : 	STRUCT
		udiCurLatchPosition : UDINT; (*色组锁标位置*)
	END_STRUCT;
	ToAsp_typ : 	STRUCT
		strDataST1 : ARRAY[0..ST_SEP_LEN_MINUS_ONE]OF STRING[ST_SEP_DATA_LEN];
		strDataST2 : ARRAY[0..ST_SEP_LEN_MINUS_ONE]OF STRING[ST_SEP_DATA_LEN];
		strDataST3 : ARRAY[0..ST_SEP_LEN_MINUS_ONE]OF STRING[ST_SEP_DATA_LEN];
		strDataST4 : ARRAY[0..ST_SEP_LEN_MINUS_ONE]OF STRING[ST_SEP_DATA_LEN];
		strDataST5 : ARRAY[0..ST_SEP_LEN_MINUS_ONE]OF STRING[ST_SEP_DATA_LEN];
		strDataST6 : ARRAY[0..ST_SEP_LEN_MINUS_ONE]OF STRING[ST_SEP_DATA_LEN];
		diWindowWidth : DINT; (*锁标窗口宽度*)
		usiCmdLatchPos : USINT; (*锁标指令*)
		udiCurLatchPosition : UDINT; (*色组锁标位置*)
		diPuWindowIntervalmm : DINT; (*当前横向自定义距离值*)
		usiActiveDrawMode : USINT; (*0-代表普通X67双光眼绘图；<br><br>
1-代表X67纵跟前横跟首模式绘图；<br><br>
2-代表X67单标记模式绘图(只画上光眼)<br><br>
3-代表X67单标记模式绘图(只画下光眼)
10-代表BST单眼模式绘图
11-代表BST双眼模式绘图*)
		diSImage : DINT; (*版周数据*)
		udiMarkSelfPosition : UDINT;
		udiMarkFirstPosition : UDINT;
		udiMarkFrontPosition : UDINT;
		usiMarkEnableBST : USINT;
	END_STRUCT;
	Asp_Interface_typ : 	STRUCT
		stFromAsp : FromAsp_typ;
		stToAsp : ToAsp_typ;
	END_STRUCT;
	ToMain_typ : 	STRUCT  (*mappView -> 后端*)
		usiActivePU : USINT; (*切换当前色组*)
		usiOneMarkMode : USINT; (*单标记开关 gSetPuOneMarkMode*)
		usiCmdLeft : USINT; (*曲线左平移*)
		usiCmdRight : USINT; (*曲线右平移*)
		usiCmdLatchPosLeft : USINT; (*锁标窗口左移*)
		usiCmdLatchPosRight : USINT; (*锁标窗口右移*)
		usiVisMarkIntervalMinus : USINT; (*横向窗口自定义距离值减小*)
		usiVisMarkIntervalAdd : USINT; (*横向窗口自定义距离值增大*)
		usiCmdLatchPos : USINT; (*锁标指令*)
		usiActivePuTeachMode : USINT; (*解锁曲线左右移动*)
		diSideFollowPu1 : DINT; (*横向跟首色开关*)
		diSideWindowDefine : DINT; (*横向窗口自定义开关*)
		diWindowWidth : DINT; (*锁标窗口宽度*)
		udiLatchPosition : ARRAY[0..12]OF UDINT; (*每一色色组锁标位置*)
	END_STRUCT;
	FromMain_typ : 	STRUCT  (*后端 -> mappView*)
		usiActiveDrawMode : USINT; (*0-普通 X67 双光眼;1-纵跟前横跟首;2-单标记模式*)
		diSImage : DINT; (*版周数据*)
		udiActivePuLatchPos : UDINT; (*当前色组锁标位置*)
		diPuWindowIntervalmm : DINT; (*当前横向自定义距离值*)
		diSideWindowInterval : ARRAY[0..12]OF DINT; (*每一色组横向距离自定义距离*)
		usiDataST1 : ARRAY[0..ST_DATA_LEN_MINUS_ONE]OF USINT; (*上光眼绘图数据*)
		usiDataST2 : ARRAY[0..ST_DATA_LEN_MINUS_ONE]OF USINT; (*下光眼绘图数据*)
		usiDataST3 : ARRAY[0..ST_DATA_LEN_MINUS_ONE]OF USINT;
		usiDataST4 : ARRAY[0..ST_DATA_LEN_MINUS_ONE]OF USINT;
		usiDataST5 : ARRAY[0..ST_DATA_LEN_MINUS_ONE]OF USINT;
		usiDataST6 : ARRAY[0..ST_DATA_LEN_MINUS_ONE]OF USINT;
		diAmrAllMarkPos : ARRAY[0..99]OF DINT; (*自动搜索搜到的有效标位置信息*)
		usiMarkSelectSelf : USINT; (*本色*)
		usiMarkSelectFront : USINT; (*前色*)
		usiMarkSelectFirst : USINT; (*首色*)
	END_STRUCT;
	Main_Interface_typ : 	STRUCT
		stFromMain : FromMain_typ;
		stToMain : ToMain_typ;
	END_STRUCT;
END_TYPE
```

### GlobalMiddle.var
```iecst
VAR
	gstHmi : HMI_Interface_typ;
	gstMiddle : Middle_Interface_typ;
	gstAspInface : Asp_Interface_typ;
	gstMainInface : Main_Interface_typ;
END_VAR
(*CONSTANT*)
VAR CONSTANT
	ST_DATA_LEN : UDINT := 1100;
	ST_DATA_LEN_MINUS_ONE : UDINT := ST_DATA_LEN-1;
	ST_DATA_LEN_DOUBLE : UDINT := ST_DATA_LEN*2;
	ST_DATA_LEN_4T3 : UDINT := ST_DATA_LEN*4/3;
	ST_SEP_DATA_LEN : UDINT := 252;
	ST_SEP_LEN : UDINT := ST_DATA_LEN_4T3/ST_SEP_DATA_LEN + 1;
	ST_SEP_LEN_MINUS_ONE : UDINT := ST_SEP_LEN-1;
	ST_PU_SIZE : UDINT := 10;
END_VAR
```

### Program Logical/LQR (ANSIC)

#### Cyclic.c - Cyclic code
```c
#include <bur/plctypes.h>

#ifdef _DEFAULT_INCLUDES
	#include <AsDefault.h>
#endif

#define LQR_STATE_COUNT_C 4
#define LQR_INPUT_COUNT_C 2
#define LQR_GAIN_STRIDE_C 4

static REAL LqrAbs(REAL value)
{
	if (value < 0.0f) {
		return -value;
	}

	return value;
}

static REAL LqrClamp(REAL value, REAL limit)
{
	if (value > limit) {
		stLqrStatus.bSaturated = 1;
		return limit;
	}
	if (value < -limit) {
		stLqrStatus.bSaturated = 1;
		return -limit;
	}

	return value;
}

static void LqrClearOutput(void)
{
	USINT i;

	for (i = 0; i < LQR_INPUT_COUNT_C; i++) {
		arLqrU[i] = 0.0f;
	}
}

static void LqrClearError(void)
{
	USINT i;

	for (i = 0; i < LQR_STATE_COUNT_C; i++) {
		arLqrError[i] = 0.0f;
	}
}

void _CYCLIC ProgramCyclic(void)
{
	USINT i;
	USINT j;
	REAL rSum;
	REAL rLimit;

	stLqrStatus.bEnabled = bLqrEnable;
	stLqrStatus.bValid = 0;
	stLqrStatus.bSaturated = 0;
	stLqrStatus.usiErrorCode = 0;

	if (bLqrReset) {
		LqrClearOutput();
		LqrClearError();
		return;
	}

	if (!bLqrEnable) {
		LqrClearOutput();
		return;
	}

	rLimit = LqrAbs(rLqrMaxAbsU);
	if (rLimit <= 0.0f) {
		LqrClearOutput();
		stLqrStatus.usiErrorCode = 1;
		return;
	}

	for (i = 0; i < LQR_STATE_COUNT_C; i++) {
		arLqrError[i] = arLqrX[i] - arLqrXRef[i];
	}

	for (j = 0; j < LQR_INPUT_COUNT_C; j++) {
		rSum = 0.0f;
		for (i = 0; i < LQR_STATE_COUNT_C; i++) {
			rSum += arLqrK[(j * LQR_GAIN_STRIDE_C) + i] * arLqrError[i];
		}
		arLqrU[j] = LqrClamp(-rSum, rLimit);
	}

	stLqrStatus.bValid = 1;
	if (stLqrStatus.bSaturated) {
		stLqrStatus.usiErrorCode = 2;
	}
}
```

#### Init.c - Initialization code
```c
#include <bur/plctypes.h>

#ifdef _DEFAULT_INCLUDES
	#include <AsDefault.h>
#endif

#define LQR_STATE_COUNT_C 4
#define LQR_INPUT_COUNT_C 2
#define LQR_GAIN_COUNT_C 8

static void LqrClearVectors(void)
{
	USINT i;

	for (i = 0; i < LQR_STATE_COUNT_C; i++) {
		arLqrX[i] = 0.0f;
		arLqrXRef[i] = 0.0f;
		arLqrError[i] = 0.0f;
	}

	for (i = 0; i < LQR_INPUT_COUNT_C; i++) {
		arLqrU[i] = 0.0f;
	}
}

static void LqrLoadDefaultGains(void)
{
	USINT i;

	for (i = 0; i < LQR_GAIN_COUNT_C; i++) {
		arLqrK[i] = 0.0f;
	}

	arLqrK[0] = 2.0f;
	arLqrK[1] = 0.4f;
	arLqrK[6] = 2.0f;
	arLqrK[7] = 0.4f;
}

void _INIT ProgramInit(void)
{
	bLqrEnable = 0;
	bLqrReset = 0;
	bLqrUseManualGains = 0;
	rLqrMaxAbsU = 100.0f;
	stLqrStatus.bEnabled = 0;
	stLqrStatus.bValid = 0;
	stLqrStatus.bSaturated = 0;
	stLqrStatus.usiErrorCode = 0;

	LqrClearVectors();
	LqrLoadDefaultGains();
}
```

#### Exit.c - Exit code
```c
#include <bur/plctypes.h>

#ifdef _DEFAULT_INCLUDES
	#include <AsDefault.h>
#endif

void _EXIT ProgramExit(void)
{
	arLqrU[0] = 0.0f;
	arLqrU[1] = 0.0f;
	stLqrStatus.bValid = 0;
}
```

#### Types.typ - Local data types
```iecst
TYPE
	LqrStatus_typ : 	STRUCT
		bEnabled : BOOL;
		bValid : BOOL;
		bSaturated : BOOL;
		usiErrorCode : USINT;
	END_STRUCT;

END_TYPE
```

#### Variables.var - Local variables
```iecst
VAR
	bLqrEnable : BOOL;
	bLqrReset : BOOL;
	bLqrUseManualGains : BOOL;
	stLqrStatus : LqrStatus_typ;
	rLqrMaxAbsU : REAL;
	arLqrX : ARRAY[0..3] OF REAL;
	arLqrXRef : ARRAY[0..3] OF REAL;
	arLqrK : ARRAY[0..7] OF REAL;
	arLqrU : ARRAY[0..1] OF REAL;
	arLqrError : ARRAY[0..3] OF REAL;
END_VAR
```

### Program Logical/SVG (ANSIC)

#### Types.typ
```iecst
TYPE
	SvgTransformField_typ : 	STRUCT
		uiOffset : UINT;
		uiLength : UINT;
	END_STRUCT;

	SvgTransformMap_typ : 	STRUCT
		stEmergencyStyle : SvgTransformField_typ;
		stLine1Duration : SvgTransformField_typ;
		stLine1Style : SvgTransformField_typ;
		stLine2Duration : SvgTransformField_typ;
		stLine2Style : SvgTransformField_typ;
		stFan1Duration : SvgTransformField_typ;
		stFan1Spin : SvgTransformField_typ;
		stRollerUpDuration : SvgTransformField_typ;
		stRollerUpTranslate : SvgTransformField_typ;
		stRollerDownStyle : SvgTransformField_typ;
		stColorBoxStyle : SvgTransformField_typ;
	END_STRUCT;

	SvgPuCommand_typ : 	STRUCT
		bEmergency : BOOL;
		bFan1Rotate : BOOL;
		bRollerUpDown : BOOL;
		bRollerDownGreen : BOOL;
		bColorBoxYellow : BOOL;
		bManualTestMode : BOOL;
	END_STRUCT;

	SvgPuText_typ : 	STRUCT
		strTemplate : STRING[1000];
		strEmergencyNormal : STRING[16];
		strEmergencyAlarm : STRING[16];
		strDisplayShow : STRING[20];
		strDisplayHide : STRING[20];
		strFan1DurationStop : STRING[8];
		strFan1DurationRun : STRING[8];
		strFan1SpinStop : STRING[16];
		strFan1SpinRun : STRING[16];
		strRollerUpDuration : STRING[8];
		strRollerUpHome : STRING[16];
		strRollerUpDown : STRING[16];
		strRollerDownNormal : STRING[16];
		strRollerDownGreen : STRING[16];
		strColorBoxNormal : STRING[16];
		strColorBoxYellow : STRING[16];
	END_STRUCT;

	SvgPuUnit_typ : 	STRUCT
		stCmd : SvgPuCommand_typ;
		stText : SvgPuText_typ;
		stMap : SvgTransformMap_typ;
		strTransform : STRING[1000];
		bTransformReady : BOOL;
	END_STRUCT;

END_TYPE
```

#### Variables.var
```iecst
VAR CONSTANT
	SVG_MAX_PU_COUNT : USINT := 8;
	SVG_MAX_PU_COUNT_MINUS_ONE : USINT := SVG_MAX_PU_COUNT - 1;
	SVG_DURATION_FIELD_LEN : USINT := 5;
	SVG_DURATION_MAX_MS : UDINT := 99999;
	SVG_FAN1_STOP_DURATION_MS : UDINT := 0;
	SVG_FAN1_RUN_DURATION_MS : UDINT := 1000;
	SVG_ROLLER_UP_DURATION_MS : UDINT := 100;
END_VAR
VAR
	strTransform : STRING[1000];
	usiSvgPuCount : USINT;
	usiActiveSvgPu : USINT;
	bRandomMotionTestMode : BOOL;
	bCmdRandomMotionOnce : BOOL;
	bOldCmdRandomMotionOnce : BOOL;
	astSvgPu : ARRAY[0..SVG_MAX_PU_COUNT_MINUS_ONE] OF SvgPuUnit_typ;
END_VAR
```

#### Cyclic.c
```c
#include <bur/plctypes.h>
#include <stdlib.h>

#ifdef _DEFAULT_INCLUDES
	#include <AsDefault.h>
#endif

#define SVG_MAX_PU_COUNT_LIMIT 8

static void SvgLoadTemplate(SvgPuUnit_typ* pPu)
{
	brsstrcpy((UDINT)pPu->strTransform, (UDINT)pPu->stText.strTemplate);
	pPu->bTransformReady = 1;
}

static void SvgCopyField(SvgPuUnit_typ* pPu, SvgTransformField_typ* pField, char* pValue)
{
	brsmemcpy((UDINT)&pPu->strTransform[pField->uiOffset], (UDINT)pValue, pField->uiLength);
}

static void SvgApplyCommands(SvgPuUnit_typ* pPu)
{
	if (pPu->stCmd.bEmergency) {
		SvgCopyField(pPu, &pPu->stMap.stEmergencyStyle, pPu->stText.strEmergencyAlarm);
	} else {
		SvgCopyField(pPu, &pPu->stMap.stEmergencyStyle, pPu->stText.strEmergencyNormal);
	}

	if (!pPu->stCmd.bRollerUpDown) {
		SvgCopyField(pPu, &pPu->stMap.stLine1Duration, pPu->stText.strRollerUpDuration);
		SvgCopyField(pPu, &pPu->stMap.stLine1Style, pPu->stText.strDisplayShow);
	} else {
		SvgCopyField(pPu, &pPu->stMap.stLine1Duration, pPu->stText.strRollerUpDuration);
		SvgCopyField(pPu, &pPu->stMap.stLine1Style, pPu->stText.strDisplayHide);
	}

	if (pPu->stCmd.bRollerUpDown) {
		SvgCopyField(pPu, &pPu->stMap.stLine2Duration, pPu->stText.strRollerUpDuration);
		SvgCopyField(pPu, &pPu->stMap.stLine2Style, pPu->stText.strDisplayShow);
	} else {
		SvgCopyField(pPu, &pPu->stMap.stLine2Duration, pPu->stText.strRollerUpDuration);
		SvgCopyField(pPu, &pPu->stMap.stLine2Style, pPu->stText.strDisplayHide);
	}

	if (pPu->stCmd.bFan1Rotate) {
		SvgCopyField(pPu, &pPu->stMap.stFan1Duration, pPu->stText.strFan1DurationRun);
		SvgCopyField(pPu, &pPu->stMap.stFan1Spin, pPu->stText.strFan1SpinRun);
	} else {
		SvgCopyField(pPu, &pPu->stMap.stFan1Duration, pPu->stText.strFan1DurationStop);
		SvgCopyField(pPu, &pPu->stMap.stFan1Spin, pPu->stText.strFan1SpinStop);
	}

	if (pPu->stCmd.bRollerUpDown) {
		SvgCopyField(pPu, &pPu->stMap.stRollerUpDuration, pPu->stText.strRollerUpDuration);
		SvgCopyField(pPu, &pPu->stMap.stRollerUpTranslate, pPu->stText.strRollerUpDown);
	} else {
		SvgCopyField(pPu, &pPu->stMap.stRollerUpDuration, pPu->stText.strRollerUpDuration);
		SvgCopyField(pPu, &pPu->stMap.stRollerUpTranslate, pPu->stText.strRollerUpHome);
	}

	if (pPu->stCmd.bRollerDownGreen) {
		SvgCopyField(pPu, &pPu->stMap.stRollerDownStyle, pPu->stText.strRollerDownGreen);
	} else {
		SvgCopyField(pPu, &pPu->stMap.stRollerDownStyle, pPu->stText.strRollerDownNormal);
	}

	if (pPu->stCmd.bColorBoxYellow) {
		SvgCopyField(pPu, &pPu->stMap.stColorBoxStyle, pPu->stText.strColorBoxYellow);
	} else {
		SvgCopyField(pPu, &pPu->stMap.stColorBoxStyle, pPu->stText.strColorBoxNormal);
	}
}

static USINT SvgGetValidPuCount(void)
{
	if (usiSvgPuCount == 0) {
		usiSvgPuCount = 1;
	}

	if (usiSvgPuCount > SVG_MAX_PU_COUNT_LIMIT) {
		usiSvgPuCount = SVG_MAX_PU_COUNT_LIMIT;
	}

	return usiSvgPuCount;
}

static USINT SvgGetActivePuIndex(USINT usiPuCount)
{
	if (usiActiveSvgPu >= usiPuCount) {
		usiActiveSvgPu = 0;
	}

	return usiActiveSvgPu;
}

static BOOL SvgRandomBool(void)
{
	return (BOOL)(rand() & 1);
}

static void SvgRandomizePu(SvgPuUnit_typ* pPu)
{
	pPu->stCmd.bManualTestMode = 0;
	pPu->stCmd.bEmergency = SvgRandomBool();
	pPu->stCmd.bFan1Rotate = SvgRandomBool();
	pPu->stCmd.bRollerUpDown = SvgRandomBool();
	pPu->stCmd.bRollerDownGreen = SvgRandomBool();
	pPu->stCmd.bColorBoxYellow = SvgRandomBool();
	pPu->bTransformReady = 0;
}

static void SvgRunRandomMotionOnce(USINT usiPuCount)
{
	USINT usiIdx;

	for (usiIdx = 0; usiIdx < usiPuCount; usiIdx++) {
		SvgRandomizePu(&astSvgPu[usiIdx]);
	}
}

void _CYCLIC ProgramCyclic(void)
{
	USINT usiIdx;
	USINT usiPuCount;
	USINT usiActiveIdx;

	usiPuCount = SvgGetValidPuCount();
	usiActiveIdx = SvgGetActivePuIndex(usiPuCount);

	if (bRandomMotionTestMode && bCmdRandomMotionOnce && !bOldCmdRandomMotionOnce) {
		SvgRunRandomMotionOnce(usiPuCount);
	}
	bOldCmdRandomMotionOnce = bCmdRandomMotionOnce;

	if (astSvgPu[usiActiveIdx].stCmd.bManualTestMode) {
		astSvgPu[usiActiveIdx].bTransformReady = 0;
		return;
	}

	for (usiIdx = 0; usiIdx < usiPuCount; usiIdx++) {
		if (!astSvgPu[usiIdx].bTransformReady) {
			SvgLoadTemplate(&astSvgPu[usiIdx]);
		}

		if (!astSvgPu[usiIdx].stCmd.bManualTestMode) {
			SvgApplyCommands(&astSvgPu[usiIdx]);
		}
	}

	brsstrcpy((UDINT)strTransform, (UDINT)astSvgPu[usiActiveIdx].strTransform);
}
```

#### Init.c
```c
#include <bur/plctypes.h>

#ifdef _DEFAULT_INCLUDES
	#include <AsDefault.h>
#endif

#define SVG_MAX_PU_COUNT_LIMIT 8

#define SVG_TEMPLATE_TEXT "[{\"select\":\"#emergency\",\"duration\":0,\"style\":\"fill:1\"},{\"select\":\"#line_1\",\"duration\": 1000,\"style\":\"display:inline\"},{\"select\":\"#line_2\",\"duration\": 1000,\"style\":\"display:inline\"},{\"select\":\"#fan1\",\"duration\":    0,\"spin\":[0,0,0]  },{\"select\":\"#roller_up\",\"duration\": 1000,\"translate\":[168, 425]},{\"select\":\"#roller_down\",\"duration\":0,\"style\":\"fill:2\"},{\"select\":\"#color_box\",\"duration\":0,\"style\":\"fill:3\"}]"

static void SvgInitField(SvgTransformField_typ* pField, UINT uiOffset, UINT uiLength)
{
	pField->uiOffset = uiOffset;
	pField->uiLength = uiLength;
}

static void SvgFormatDuration(char* pDest, UDINT udiDuration)
{
	INT iPos;
	UDINT udiValue;

	udiValue = udiDuration;
	if (udiValue > SVG_DURATION_MAX_MS) {
		udiValue = SVG_DURATION_MAX_MS;
	}

	for (iPos = 0; iPos < SVG_DURATION_FIELD_LEN; iPos++) {
		pDest[iPos] = ' ';
	}
	pDest[SVG_DURATION_FIELD_LEN] = '\0';

	iPos = SVG_DURATION_FIELD_LEN - 1;
	do {
		pDest[iPos] = (char)('0' + (udiValue % 10));
		udiValue = udiValue / 10;
		iPos--;
	} while (udiValue > 0 && iPos >= 0);
}

static void SvgInitPuUnit(SvgPuUnit_typ* pPu)
{
	pPu->stCmd.bEmergency = 0;
	pPu->stCmd.bFan1Rotate = 0;
	pPu->stCmd.bRollerUpDown = 0;
	pPu->stCmd.bRollerDownGreen = 0;
	pPu->stCmd.bColorBoxYellow = 0;
	pPu->stCmd.bManualTestMode = 0;

	brsstrcpy((UDINT)pPu->stText.strTemplate, (UDINT)SVG_TEMPLATE_TEXT);
	brsstrcpy((UDINT)pPu->stText.strEmergencyNormal, (UDINT)"fill:1");
	brsstrcpy((UDINT)pPu->stText.strEmergencyAlarm, (UDINT)"fill:3");
	brsstrcpy((UDINT)pPu->stText.strDisplayShow, (UDINT)"display:inline");
	brsstrcpy((UDINT)pPu->stText.strDisplayHide, (UDINT)"display:none  ");
	SvgFormatDuration(pPu->stText.strFan1DurationStop, SVG_FAN1_STOP_DURATION_MS);
	SvgFormatDuration(pPu->stText.strFan1DurationRun, SVG_FAN1_RUN_DURATION_MS);
	brsstrcpy((UDINT)pPu->stText.strFan1SpinStop, (UDINT)"[0,0,0]  ");
	brsstrcpy((UDINT)pPu->stText.strFan1SpinRun, (UDINT)"[360,0,0]");
	SvgFormatDuration(pPu->stText.strRollerUpDuration, SVG_ROLLER_UP_DURATION_MS);
	brsstrcpy((UDINT)pPu->stText.strRollerUpHome, (UDINT)"[168, 425]");
	brsstrcpy((UDINT)pPu->stText.strRollerUpDown, (UDINT)"[168, 470]");
	brsstrcpy((UDINT)pPu->stText.strRollerDownNormal, (UDINT)"fill:2");
	brsstrcpy((UDINT)pPu->stText.strRollerDownGreen, (UDINT)"fill:1");
	brsstrcpy((UDINT)pPu->stText.strColorBoxNormal, (UDINT)"fill:3");
	brsstrcpy((UDINT)pPu->stText.strColorBoxYellow, (UDINT)"fill:0");

	SvgInitField(&pPu->stMap.stEmergencyStyle, 46, 6);
	SvgInitField(&pPu->stMap.stLine1Duration, 86, SVG_DURATION_FIELD_LEN);
	SvgInitField(&pPu->stMap.stLine1Style, 101, 14);
	SvgInitField(&pPu->stMap.stLine2Duration, 149, SVG_DURATION_FIELD_LEN);
	SvgInitField(&pPu->stMap.stLine2Style, 164, 14);
	SvgInitField(&pPu->stMap.stFan1Duration, 210, SVG_DURATION_FIELD_LEN);
	SvgInitField(&pPu->stMap.stFan1Spin, 223, 9);
	SvgInitField(&pPu->stMap.stRollerUpDuration, 268, SVG_DURATION_FIELD_LEN);
	SvgInitField(&pPu->stMap.stRollerUpTranslate, 286, 10);
	SvgInitField(&pPu->stMap.stRollerDownStyle, 345, 6);
	SvgInitField(&pPu->stMap.stColorBoxStyle, 399, 6);

	brsstrcpy((UDINT)pPu->strTransform, (UDINT)"");
	pPu->bTransformReady = 0;
}

void _INIT ProgramInit(void)
{
	USINT usiIdx;

	brsstrcpy((UDINT)strTransform, (UDINT)"");
	usiSvgPuCount = 1;
	usiActiveSvgPu = 0;
	bRandomMotionTestMode = 0;
	bCmdRandomMotionOnce = 0;
	bOldCmdRandomMotionOnce = 0;

	for (usiIdx = 0; usiIdx < SVG_MAX_PU_COUNT_LIMIT; usiIdx++) {
		SvgInitPuUnit(&astSvgPu[usiIdx]);
	}
}
```

#### manual_test_commands.txt
```
Manual Paper transform test commands
====================================

Write any one of these complete JSON strings to SVG:strTransform for a single-part test.
Set SVG:astSvgPu[0].stCmd.bManualTestMode = 1 before writing these commands, otherwise ProgramCyclic will overwrite strTransform.
Set SVG:astSvgPu[0].stCmd.bManualTestMode = 0 to return to automatic command-bit control.

1. emergency - red  修改
[{"select":"#emergency","duration":0,"style":"fill:3"}]

2. emergency - normal gray  修改
[{"select":"#emergency","duration":0,"style":"fill:1"}]

3. line_1 - show 通过
[{"select":"#line_1","duration":0,"style":"display:inline"}]

4. line_1 - hide 通过
[{"select":"#line_1","duration":0,"style":"display:none"}]

5. line_2 - show  通过
[{"select":"#line_2","duration":0,"style":"display:inline"}]

6. line_2 - hide 通过
[{"select":"#line_2","duration":0,"style":"display:none"}]

7. fan1 - rotate once around local center (0,0)   通过
[{"select":"#fan1","duration":1000,"spin":[360,0,0]}]

8. fan1 - stop/no rotation command   通过
[{"select":"#fan1","duration":0,"spin":[0,0,0]}]

9. roller_up - move down 20 units 修改
[{"select":"#roller_up","duration":1000,"translate":[168, 470]}]

10. roller_up - return home 修改
[{"select":"#roller_up","duration":1000,"translate":[168, 425]}]

11. roller_down - green outline 修改
[{"select":"#roller_down","duration":0,"style":"fill:1"}]

12. roller_down - normal 修改
[{"select":"#roller_down","duration":0,"style":"fill:2"}]

13. color_box - yellow 修改
[{"select":"#color_box","duration":0,"style":"fill:0"}]

14. color_box - normal 修改
[{"select":"#color_box","duration":0,"style":"fill:3"}]

15. all active  (根据以上修改)
[{"select":"#emergency","duration":0,"style":"fill:#ff0000"},{"select":"#line_1","duration":0,"style":"display:none"},{"select":"#line_2","duration":0,"style":"display:none"},{"select":"#fan1","duration":1000,"spin":[360,0,0]},{"select":"#roller_up","duration":1000,"translate":[0,20]},{"select":"#roller_down","duration":0,"style":"fill:url(#circleGrad);stroke:#00c853;stroke-width:5px"},{"select":"#color_box","duration":0,"style":"fill:#ffd400"}]

16. all normal （根据以上修改）
[{"select":"#emergency","duration":0,"style":"fill:#9d9d9d"},{"select":"#line_1","duration":0,"style":"display:inline"},{"select":"#line_2","duration":0,"style":"display:inline"},{"select":"#fan1","duration":0,"spin":[0,0,0]},{"select":"#roller_up","duration":1000,"translate":[0,0]},{"select":"#roller_down","duration":0,"style":"fill:url(#circleGrad);stroke:#777777;stroke-width:0px"},{"select":"#color_box","duration":0,"style":"fill:#d2d2d2"}]
```

Listed in the project but not available here: Logical/Global.typ, Logical/Global.var, Logical/Middleware/MidTrans/Types.typ
